Omron CX-Programmer project NuevoProyecto (CX-Programmer 9.31)

# PLC NuevoPLC1: CJ1M CPU11

## Program NuevoPrograma1 (cyclic task 0)
; La v1.1 funciona correctament la inicialitzacio, manual(La linea 1 del E_F4 te un SMM ja que sino al sortir es mantidria EM_0 en on)
Local symbols
C1_BE 0.07 BOOL  ; Bolet de emergencia
C1_COM1_FI_CUA W511.02 BOOL  ; CUADRAT  COMPLETS COMANDA 1
C1_COM1_FI_PEN W511.03 BOOL  ; PENTAGO COMPLETS COMANDA 1
C1_COM1_FI_ROD W511.01 BOOL  ; RODONA COMPLETS COMANDA 1
C1_COM1_FI_TRI W511.00 BOOL  ; TRIANGLES COMPLETS COMANDA 1
C1_COM2_FI_CUA W511.06 BOOL  ; CUADRAT COMPLETS COMANDA 2
C1_COM2_FI_PEN W511.07 BOOL  ; PENTAGON COMPLETS COMANDA 2
C1_COM2_FI_ROD W511.05 BOOL  ; RODONA COMPLETS COMANDA 2
C1_COM2_FI_TRI W511.04 BOOL  ; TRIANGLES COMPLETS COMANDA 2
C1_DET1 0.09 BOOL  ; Detector 1 cinta 1
C1_DET2 0.08 BOOL  ; Detector 2 cinta 1
C1_DET3 0.10 BOOL  ; Detector 3 cinta 1
C1_DET4 0.11 BOOL  ; Detector 4 cinta 1
C1_EA_0 W300.00 BOOL  ; Etapa automatic 0
C1_EA_1 W300.01 BOOL  ; Etapa automatica 1 MFW
C1_EA_10 W300.10 BOOL  ; COMANDA 2 TRIANGLE ++
C1_EA_11 W300.11 BOOL  ; TRIANGLE A REBUIG
C1_EA_18 W300.12 BOOL  ; Etapa automatica 18 cuadrat
C1_EA_19 W300.13 BOOL  ; COMANDA 1 CUADRAT ++
C1_EA_2 W300.02 BOOL  ; Etapa automatica 2 T1
C1_EA_20 W300.14 BOOL  ; COMANDA 2 CUADRAT ++
C1_EA_21 W300.15 BOOL  ; CUADRAT REBUIG
C1_EA_28 W301.00 BOOL  ; ETAPA AUTOMATIC 28 PENTAGON
C1_EA_29 W301.01 BOOL  ; COMANDA 1 PENTAGON ++
C1_EA_3 W300.03 BOOL  ; Etapa automatica 3 MOFF
C1_EA_30 W301.02 BOOL  ; COMANDA 2 PENTAGON++
C1_EA_31 W301.03 BOOL  ; PENTAGON REBUIG
C1_EA_38 W301.04 BOOL  ; ESTAPA AUTOMATIC 38 RODONA
C1_EA_39 W301.05 BOOL  ; COMANDA 1 RODONA ++
C1_EA_4 W300.04 BOOL  ; Etapa automatica 4 NO EVA 1
C1_EA_40 W301.06 BOOL  ; COMANDA 2 RODONA ++
C1_EA_41 W301.07 BOOL  ; RODONA REBUIG
C1_EA_42 W301.08 BOOL  ; FI CICLE
C1_EA_5 W300.05 BOOL  ; Etapa automatica 5 OK EVA
C1_EA_6 W300.06 BOOL  ; Etapa automatica 6 T2
C1_EA_7 W300.07 BOOL  ; Etapa automatica DET4
C1_EA_8 W300.08 BOOL  ; Etapa automatica 8 Triangle
C1_EA_9 W300.09 BOOL  ; COMANDA 1 TRIANGLE++
C1_EM_0 W200.00 BOOL  ; Etapa 0 Manual
C1_EM_1 W200.01 BOOL  ; Etapa Manual1-Motor Forware
C1_EM_2 W200.02 BOOL  ; Etapa Manual2-Motor Reware
C1_EM_3 W200.03 BOOL  ; Etapa manual 3 - Aturada motor
C1_E_A1 W400.00 BOOL
C1_E_A2 W400.03 BOOL  ; Parada solicitud final de cicle
C1_E_D1 W400.05 BOOL  ; Parada de emergencia
C1_E_D3 W400.06 BOOL  ; Parada postemergencia
C1_E_F1 W400.01 BOOL  ; Produccio normal
C1_E_F4 W400.02 BOOL  ; Marcha de verificacio sense ordre
C1_E_F41 W400.04 BOOL  ; Etapa de pas Sortida Manual
C1_E_F6 W400.07 BOOL  ; Teach Marxa de Test
C1_E_F61 W400.08 BOOL  ; Teach 2
C1_HMI_A1 W103.00 BOOL  ; HABILITACIO A SCADA DE E_A1
C1_HMI_A6 W103.03 BOOL  ; HABILITACIO A SCADA DE A6
C1_HMI_COM1_PEN W14 CHANNEL  ; ENVIA EL ESTAT DE PENTAGON DE COMANDA 1
C1_HMI_COM1_QUA W12 CHANNEL  ; ENVIA EL ESTAT DE CUADRATS DE COMANDA 1
C1_HMI_COM1_ROD W13 CHANNEL  ; ENVIA EL ESTAT DE RODONES DE COMANDA 1
C1_HMI_COM1_TRI W11 CHANNEL  ; ENVIA EL ESTAT DE TRIANGLES DE COMANDA 1
C1_HMI_COM2_PEN W18 CHANNEL  ; ENVIA EL ESTAT DE PENTAGO  DE COMANDA 2
C1_HMI_COM2_QUA W16 CHANNEL  ; ENVIA EL ESTAT DE CUADRAT DE COMANDA 2
C1_HMI_COM2_ROD W17 CHANNEL  ; ENVIA EL ESTAT DE RODONA DE COMANDA 2
C1_HMI_COM2_TRI W15 CHANNEL  ; ENVIA EL ESTAT DE TRIANGLES DE COMANDA 2
C1_HMI_D2 W103.04 BOOL  ; HABILITACIO A SCADA DE D1
C1_HMI_EMER_FIS W101.03 BOOL  ; AVIS DE CINTA DE EMERGENCIA FISICA
C1_HMI_EMER_LOG W101.02 BOOL  ; AVIS CINTA DE EMERGENCIA LOGICA
C1_HMI_F1 W103.01 BOOL  ; HABILITACIO A SCADA DE F1
C1_HMI_F4 W103.02 BOOL  ; HABILITACIO A SCADA DE F4
C1_HMI_MOT_OK W101.00 BOOL  ; AVIS A LA HMI QUE LA CINTA FUNCIONA
C1_HMI_PR W101.04 BOOL  ; AVIS DEL POLSADOR DE REARME A HMI
C1_H_AMB 1.09 BOOL
C1_H_AUTO 1.03 BOOL
C1_H_MANUAL 1.04 BOOL
C1_H_ROJ 1.10 BOOL
C1_H_TEACH 1.05 BOOL
C1_H_VER 1.08 BOOL
C1_JFW 0.06 BOOL  ; Joystick Forware
C1_JRW 0.05 BOOL  ; Joystick Reward
C1_KA10 1.07 BOOL
C1_KA9 1.06 BOOL
C1_MF W201.00 BOOL  ; Marca First scan
C1_MFW 1.01 BOOL  ; Motor Forward
C1_MM W100.15 BOOL  ; Marca marxa
C1_MPP W201.04 BOOL  ; MARCA DE PARO
C1_MRW 1.00 BOOL  ; Motor Reward
C1_NOK_EVA W501.00 BOOL  ; Foto erronea
C1_OK_EVA 500.02 BOOL  ; Foto correcta
C1_PM 0.02 BOOL  ; Polsador marxa
C1_PP 0.03 BOOL  ; Polsador paro
C1_PR 0.04 BOOL  ; Polsador rearme
C1_REP W501.01 BOOL  ; Repetir foto
C1_SM1 0.00 BOOL  ; Selector de mode Pos.1
C1_SM2 0.01 BOOL  ; Selector de mode Pos.2
C1_SMA W201.01 BOOL  ; Marca selector automatic
C1_SMM 201.02 BOOL  ; Marca selector manual
C1_SMT 201.03 BOOL  ; Marca selector Teach
C1_TEACH_OK H0.00 BOOL  ; Captura correcte peça
C2_FI_CICLE 3101.00 BOOL
C2_MAGATZEM_1_3 3100.00 BOOL
C2_MAGATZEM_2_4 3100.01 BOOL
COMP_PEN1 W100.04 BOOL  ; COMPARA PENTAGONS COM1
COMP_PEN2 W100.05 BOOL  ; COMPARA PENTAGONS COM2
COMP_QUA1 W100.02 BOOL  ; COMPARA QUADRATS COM1
COMP_QUA2 W100.03 BOOL  ; COMPARA QUADRATS COM2
COMP_ROD1 W100.06 BOOL  ; COMPARA RODONES COM1
COMP_ROD2 W100.07 BOOL  ; COMPARA RODONES COM2
COMP_TRI1 W100.00 BOOL  ; COMPARA TRIANGLES COM1
COMP_TRI2 W100.01 BOOL  ; COMPARA TRIANGLES COM2
CUA_COM1 W305.02 BOOL
CUA_COM2 W305.03 BOOL
EVA_CUADRAT W510.01 BOOL  ; Foto per EVA=CUADRAT
EVA_ENABLE 510.04 BOOL  ; ACTIVAR EVA
EVA_PENTAGON W510.03 BOOL  ; Foto per EVA=PENTAGON
EVA_RODONA W510.02 BOOL  ; Foto per EVA=RODONA
EVA_TRIANGLE W510.00 BOOL  ; Foto per EVA=TRIANGLE
HMI_BE W101.05 BOOL  ; BOLET DE EMERGENCIA HMI
HMI_C1_COM1_OK W101.13 BOOL  ; VALIDACIO COM 1
HMI_C1_COM2_OK W101.14 BOOL  ; VALIDACIO COM2
HMI_C1_JF W101.08 BOOL  ; HMI C1 JOYSTICKDRETA
HMI_C1_JR W101.09 BOOL  ; HMI C1 JOYSTIC REWARD
HMI_C1_PSW W101.15 BOOL  ; PASSWORD OK
HMI_C1_Q_NO W102.01 BOOL  ; RESPOSTA NEGATIVA A ACABAR CICLE
HMI_C1_Q_SI W102.00 BOOL  ; RESPOSTA AFIRMATIVA A ACABAR CICLE
HMI_C1_TEMP_DET3 W10 UINT_BCD  ; TEMPORITZADOR DET3-DET4
HMI_C1_TEMP_EVA W9 UINT_BCD  ; TEMPORTIZADOR EVA
HMI_COM1_CUA W1 CHANNEL  ; DEMANDA DE CUADRATS PER COMANDA 1
HMI_COM1_PEN W2 CHANNEL  ; DEMANDA DE PENTAGON PER COMANDA 1
HMI_COM1_ROD W3 CHANNEL  ; DEMANDA DE RODONA PER COMANDA 1
HMI_COM1_TRI W4 CHANNEL  ; DEMANDA DE TRIANGLE PER COMANDA 1
HMI_COM2_CUA W5 CHANNEL  ; DEMANDA DE CUADRATS PER COMANDA 2
HMI_COM2_PEN W6 CHANNEL  ; DEMANDA DE PENTAGON PER COMANDA 2
HMI_COM2_ROD W7 CHANNEL  ; DEMANDA DE RODONA PER COMANDA 2
HMI_COM2_TRI W8 CHANNEL  ; DEMANDA DE TRIANGLE PER COMANDA 2
HMI_EMER_OK W101.12 BOOL  ; Validacio de emerencies
HMI_PM W101.07 BOOL  ; Polsador de marxa des de HMI
HMI_PP W101.06 BOOL  ; Polsador de paro des de HMI
MAN_FWD W201.02 BOOL  ; MOTOR FORDWARD MANUAL
MAN_RWD W201.03 BOOL  ; MOTOR REWARD MANUAL
PEN_COM1 W305.04 BOOL
PEN_COM2 W305.05 BOOL
ROD_COM1 W305.06 BOOL
ROD_COM2 W305.07 BOOL
TRI_COM1 W305.00 BOOL
TRI_COM2 W305.01 BOOL

### Section INICIALITZACIÓ_I_ETAPA_ACTIVA_GEMMA

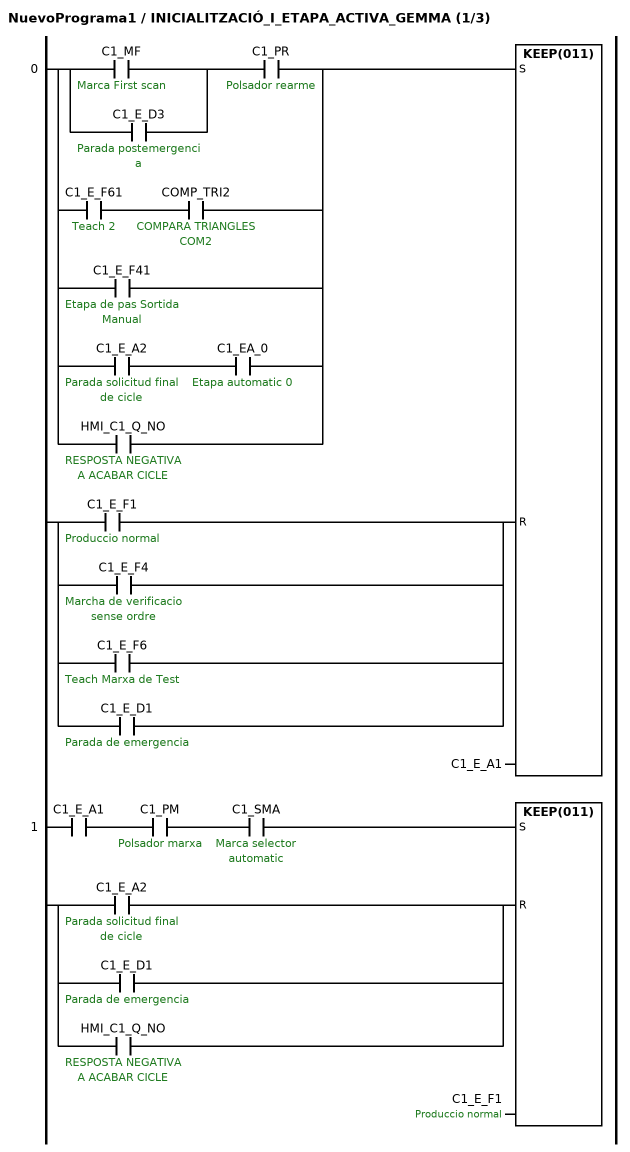
; rung 0
LD C1_MF  ; Marca First scan
OR C1_E_D3  ; Parada postemergencia
AND C1_PR  ; Polsador rearme
LD C1_E_F61  ; Teach 2
AND COMP_TRI2  ; COMPARA TRIANGLES COM2
ORLD
OR C1_E_F41  ; Etapa de pas Sortida Manual
LD C1_E_A2  ; Parada solicitud final de cicle
AND C1_EA_0  ; Etapa automatic 0
ORLD
OR HMI_C1_Q_NO  ; RESPOSTA NEGATIVA A ACABAR CICLE
LD C1_E_F1  ; Produccio normal
OR C1_E_F4  ; Marcha de verificacio sense ordre
OR C1_E_F6  ; Teach Marxa de Test
OR C1_E_D1  ; Parada de emergencia
KEEP(011) C1_E_A1
; rung 1
LD C1_E_A1
AND C1_PM  ; Polsador marxa
AND C1_SMA  ; Marca selector automatic
LD C1_E_A2  ; Parada solicitud final de cicle
OR C1_E_D1  ; Parada de emergencia
OR HMI_C1_Q_NO  ; RESPOSTA NEGATIVA A ACABAR CICLE
KEEP(011) C1_E_F1  ; Produccio normal

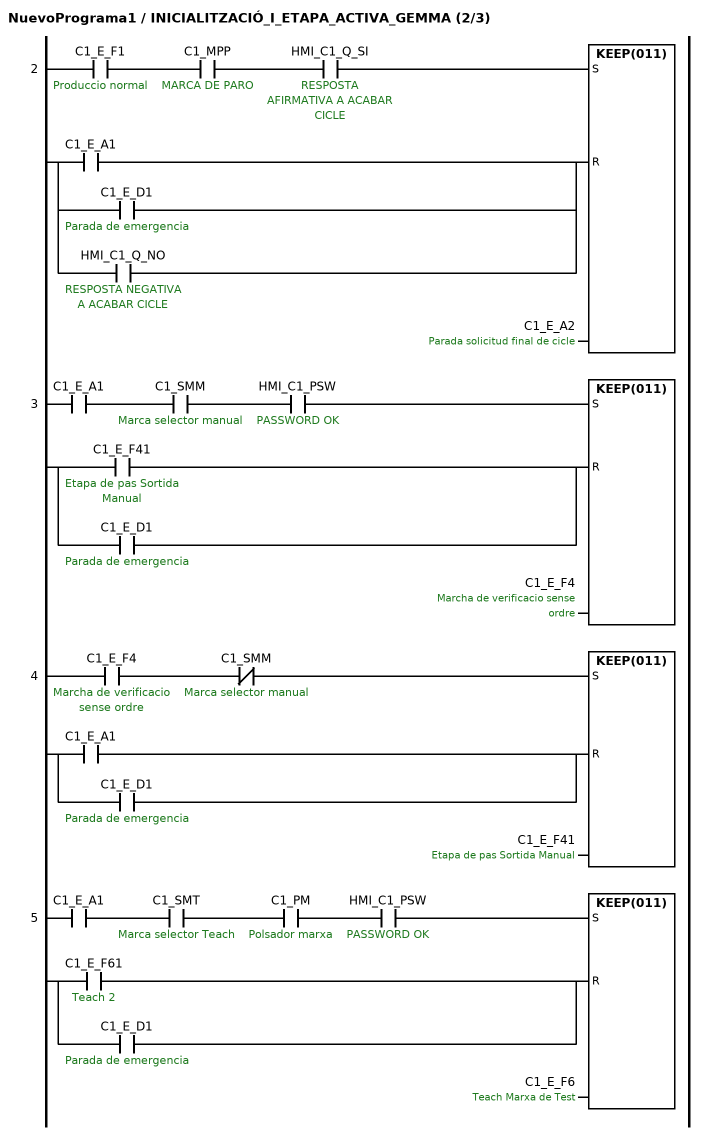
; rung 2
LD C1_E_F1  ; Produccio normal
AND C1_MPP  ; MARCA DE PARO
AND HMI_C1_Q_SI  ; RESPOSTA AFIRMATIVA A ACABAR CICLE
LD C1_E_A1
OR C1_E_D1  ; Parada de emergencia
OR HMI_C1_Q_NO  ; RESPOSTA NEGATIVA A ACABAR CICLE
KEEP(011) C1_E_A2  ; Parada solicitud final de cicle
; rung 3
LD C1_E_A1
AND C1_SMM  ; Marca selector manual
AND HMI_C1_PSW  ; PASSWORD OK
LD C1_E_F41  ; Etapa de pas Sortida Manual
OR C1_E_D1  ; Parada de emergencia
KEEP(011) C1_E_F4  ; Marcha de verificacio sense ordre
; rung 4
LD C1_E_F4  ; Marcha de verificacio sense ordre
ANDNOT C1_SMM  ; Marca selector manual
LD C1_E_A1
OR C1_E_D1  ; Parada de emergencia
KEEP(011) C1_E_F41  ; Etapa de pas Sortida Manual
; rung 5
LD C1_E_A1
AND C1_SMT  ; Marca selector Teach
AND C1_PM  ; Polsador marxa
AND HMI_C1_PSW  ; PASSWORD OK
LD C1_E_F61  ; Teach 2
OR C1_E_D1  ; Parada de emergencia
KEEP(011) C1_E_F6  ; Teach Marxa de Test

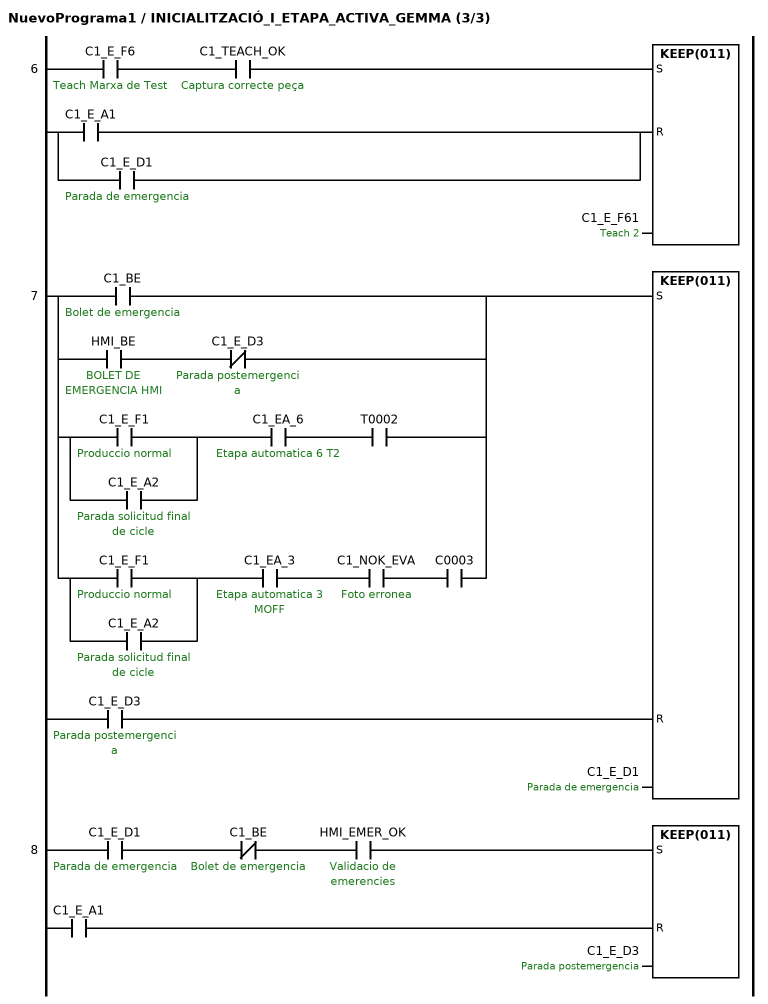
; rung 6
LD C1_E_F6  ; Teach Marxa de Test
AND C1_TEACH_OK  ; Captura correcte peça
LD C1_E_A1
OR C1_E_D1  ; Parada de emergencia
KEEP(011) C1_E_F61  ; Teach 2
; rung 7
LD C1_BE  ; Bolet de emergencia
LD HMI_BE  ; BOLET DE EMERGENCIA HMI
ANDNOT C1_E_D3  ; Parada postemergencia
ORLD
LD C1_E_F1  ; Produccio normal
OR C1_E_A2  ; Parada solicitud final de cicle
AND C1_EA_6  ; Etapa automatica 6 T2
AND T0002
ORLD
LD C1_E_F1  ; Produccio normal
OR C1_E_A2  ; Parada solicitud final de cicle
AND C1_EA_3  ; Etapa automatica 3 MOFF
AND C1_NOK_EVA  ; Foto erronea
AND C0003
ORLD
LD C1_E_D3  ; Parada postemergencia
KEEP(011) C1_E_D1  ; Parada de emergencia
; rung 8
LD C1_E_D1  ; Parada de emergencia
ANDNOT C1_BE  ; Bolet de emergencia
AND HMI_EMER_OK  ; Validacio de emerencies
LD C1_E_A1
KEEP(011) C1_E_D3  ; Parada postemergencia

### Section ACCIONS_GEMMA

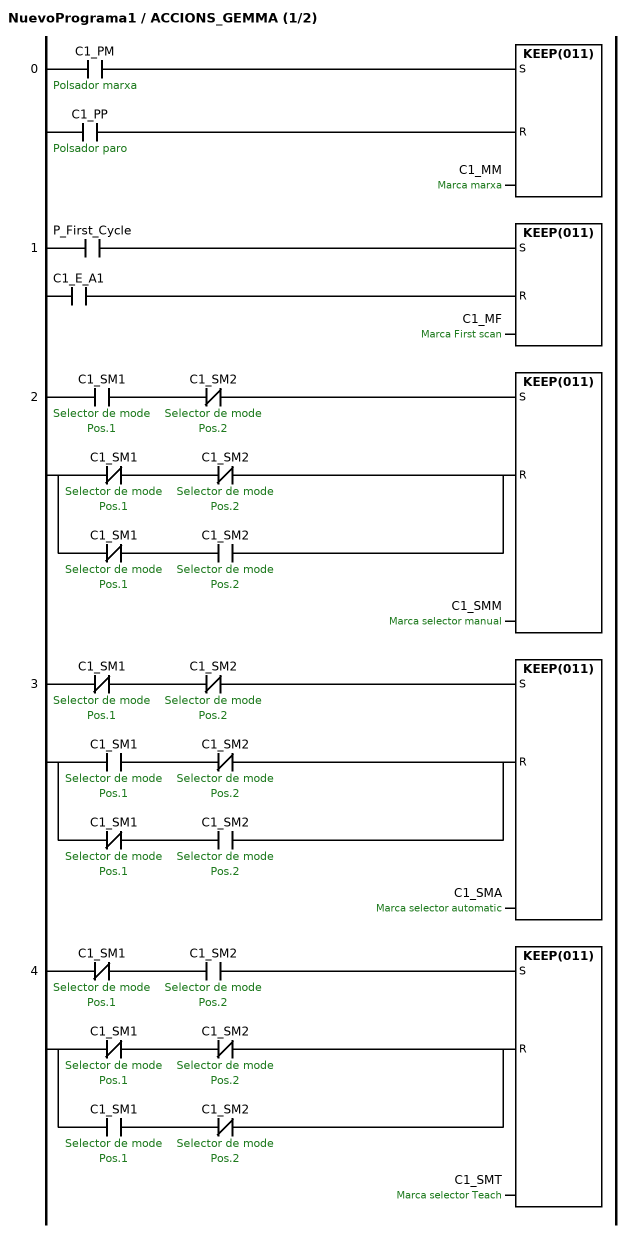
; rung 0
LD C1_PM  ; Polsador marxa
LD C1_PP  ; Polsador paro
KEEP(011) C1_MM  ; Marca marxa
; rung 1
LD P_First_Cycle
LD C1_E_A1
KEEP(011) C1_MF  ; Marca First scan
; rung 2
LD C1_SM1  ; Selector de mode Pos.1
ANDNOT C1_SM2  ; Selector de mode Pos.2
LDNOT C1_SM1  ; Selector de mode Pos.1
ANDNOT C1_SM2  ; Selector de mode Pos.2
LDNOT C1_SM1  ; Selector de mode Pos.1
AND C1_SM2  ; Selector de mode Pos.2
ORLD
KEEP(011) C1_SMM  ; Marca selector manual
; rung 3
LDNOT C1_SM1  ; Selector de mode Pos.1
ANDNOT C1_SM2  ; Selector de mode Pos.2
LD C1_SM1  ; Selector de mode Pos.1
ANDNOT C1_SM2  ; Selector de mode Pos.2
LDNOT C1_SM1  ; Selector de mode Pos.1
AND C1_SM2  ; Selector de mode Pos.2
ORLD
KEEP(011) C1_SMA  ; Marca selector automatic
; rung 4
LDNOT C1_SM1  ; Selector de mode Pos.1
AND C1_SM2  ; Selector de mode Pos.2
LDNOT C1_SM1  ; Selector de mode Pos.1
ANDNOT C1_SM2  ; Selector de mode Pos.2
LD C1_SM1  ; Selector de mode Pos.1
ANDNOT C1_SM2  ; Selector de mode Pos.2
ORLD
KEEP(011) C1_SMT  ; Marca selector Teach

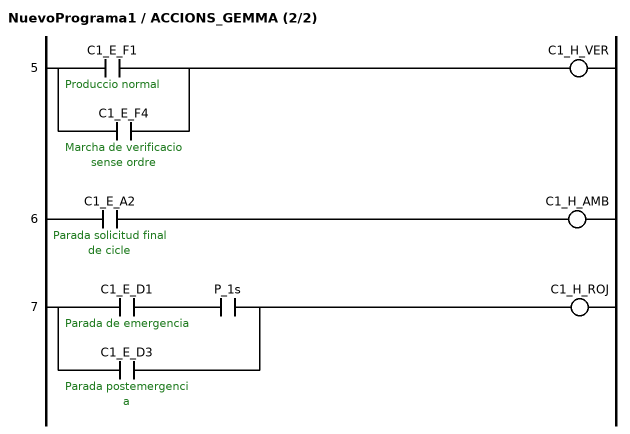
; rung 5
LD C1_E_F1  ; Produccio normal
OR C1_E_F4  ; Marcha de verificacio sense ordre
OUT C1_H_VER
; rung 6
LD C1_E_A2  ; Parada solicitud final de cicle
OUT C1_H_AMB
; rung 7
LD C1_E_D1  ; Parada de emergencia
AND P_1s
OR C1_E_D3  ; Parada postemergencia
OUT C1_H_ROJ

### Section E_F1

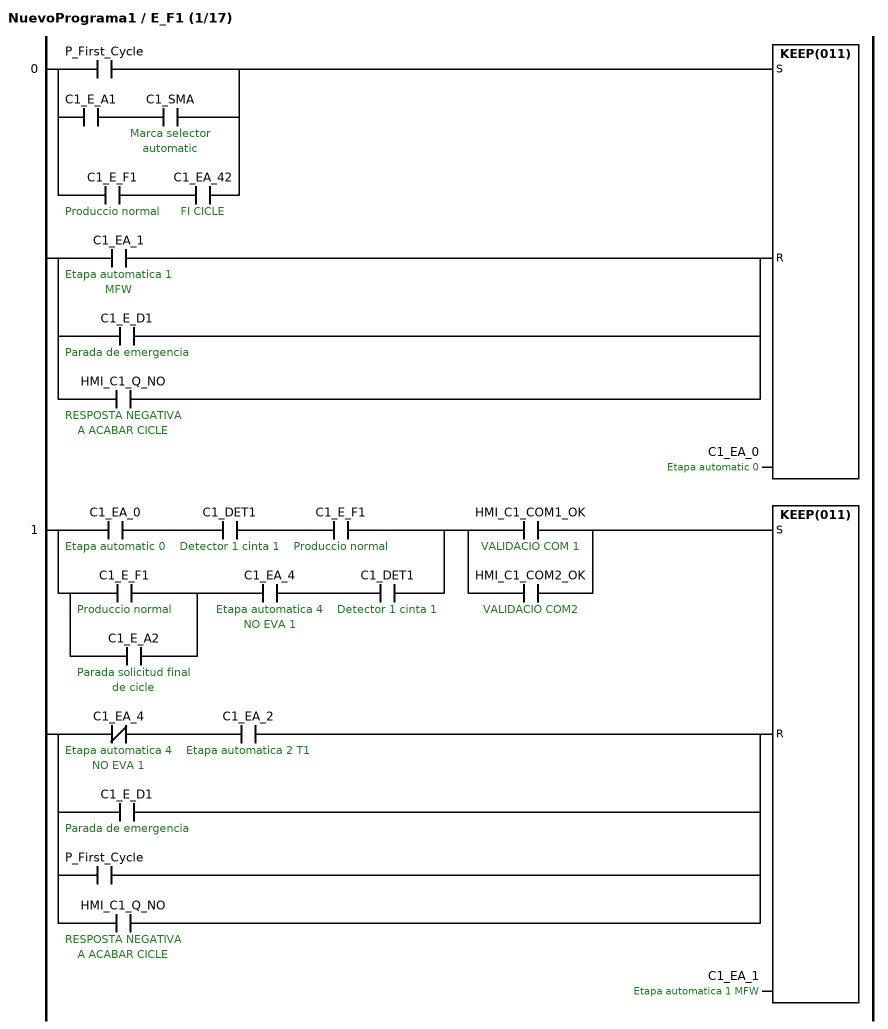
; rung 0
LD P_First_Cycle
LD C1_E_A1
AND C1_SMA  ; Marca selector automatic
ORLD
LD C1_E_F1  ; Produccio normal
AND C1_EA_42  ; FI CICLE
ORLD
LD C1_EA_1  ; Etapa automatica 1 MFW
OR C1_E_D1  ; Parada de emergencia
OR HMI_C1_Q_NO  ; RESPOSTA NEGATIVA A ACABAR CICLE
KEEP(011) C1_EA_0  ; Etapa automatic 0
; rung 1
LD C1_EA_0  ; Etapa automatic 0
AND C1_DET1  ; Detector 1 cinta 1
AND C1_E_F1  ; Produccio normal
LD C1_E_F1  ; Produccio normal
OR C1_E_A2  ; Parada solicitud final de cicle
AND C1_EA_4  ; Etapa automatica 4 NO EVA 1
AND C1_DET1  ; Detector 1 cinta 1
ORLD
LD HMI_C1_COM1_OK  ; VALIDACIO COM 1
OR HMI_C1_COM2_OK  ; VALIDACIO COM2
ANDLD
LDNOT C1_EA_4  ; Etapa automatica 4 NO EVA 1
AND C1_EA_2  ; Etapa automatica 2 T1
OR C1_E_D1  ; Parada de emergencia
OR P_First_Cycle
OR HMI_C1_Q_NO  ; RESPOSTA NEGATIVA A ACABAR CICLE
KEEP(011) C1_EA_1  ; Etapa automatica 1 MFW

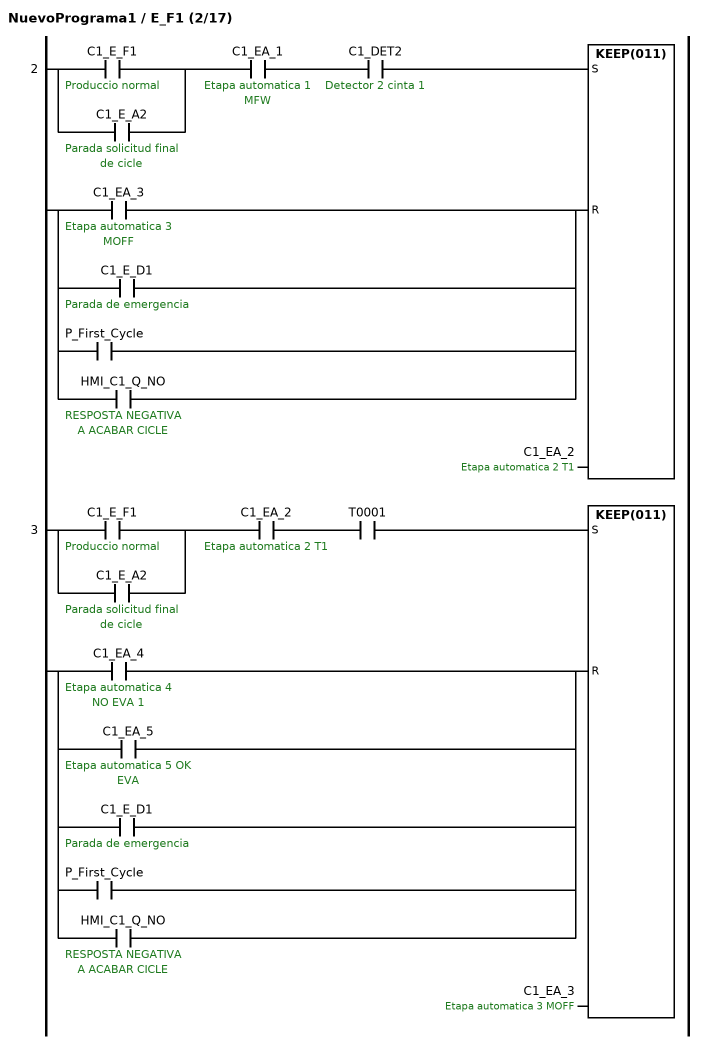
; rung 2
LD C1_E_F1  ; Produccio normal
OR C1_E_A2  ; Parada solicitud final de cicle
AND C1_EA_1  ; Etapa automatica 1 MFW
AND C1_DET2  ; Detector 2 cinta 1
LD C1_EA_3  ; Etapa automatica 3 MOFF
OR C1_E_D1  ; Parada de emergencia
OR P_First_Cycle
OR HMI_C1_Q_NO  ; RESPOSTA NEGATIVA A ACABAR CICLE
KEEP(011) C1_EA_2  ; Etapa automatica 2 T1
; rung 3
LD C1_E_F1  ; Produccio normal
OR C1_E_A2  ; Parada solicitud final de cicle
AND C1_EA_2  ; Etapa automatica 2 T1
AND T0001
LD C1_EA_4  ; Etapa automatica 4 NO EVA 1
OR C1_EA_5  ; Etapa automatica 5 OK EVA
OR C1_E_D1  ; Parada de emergencia
OR P_First_Cycle
OR HMI_C1_Q_NO  ; RESPOSTA NEGATIVA A ACABAR CICLE
KEEP(011) C1_EA_3  ; Etapa automatica 3 MOFF

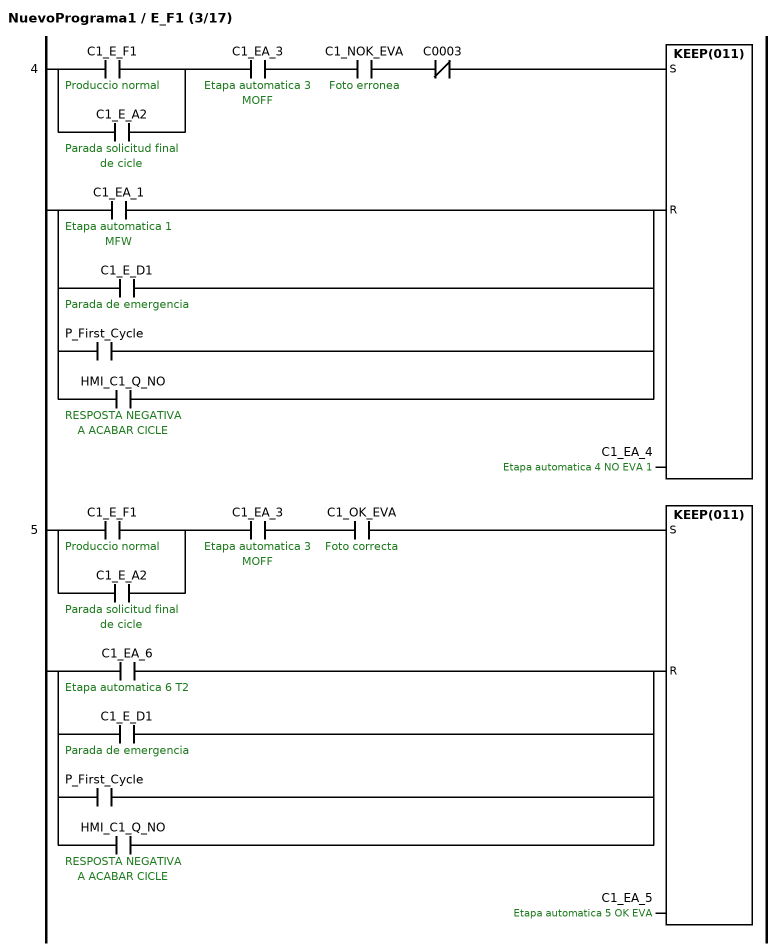
; rung 4
LD C1_E_F1  ; Produccio normal
OR C1_E_A2  ; Parada solicitud final de cicle
AND C1_EA_3  ; Etapa automatica 3 MOFF
AND C1_NOK_EVA  ; Foto erronea
ANDNOT C0003
LD C1_EA_1  ; Etapa automatica 1 MFW
OR C1_E_D1  ; Parada de emergencia
OR P_First_Cycle
OR HMI_C1_Q_NO  ; RESPOSTA NEGATIVA A ACABAR CICLE
KEEP(011) C1_EA_4  ; Etapa automatica 4 NO EVA 1
; rung 5
LD C1_E_F1  ; Produccio normal
OR C1_E_A2  ; Parada solicitud final de cicle
AND C1_EA_3  ; Etapa automatica 3 MOFF
AND C1_OK_EVA  ; Foto correcta
LD C1_EA_6  ; Etapa automatica 6 T2
OR C1_E_D1  ; Parada de emergencia
OR P_First_Cycle
OR HMI_C1_Q_NO  ; RESPOSTA NEGATIVA A ACABAR CICLE
KEEP(011) C1_EA_5  ; Etapa automatica 5 OK EVA

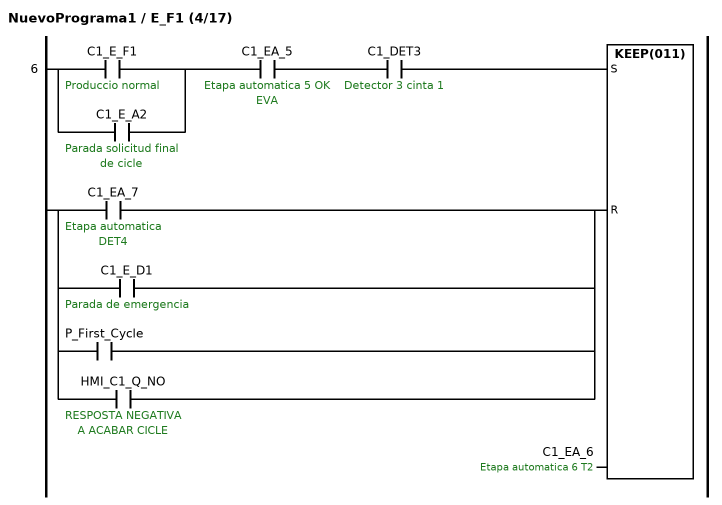
; rung 6
LD C1_E_F1  ; Produccio normal
OR C1_E_A2  ; Parada solicitud final de cicle
AND C1_EA_5  ; Etapa automatica 5 OK EVA
AND C1_DET3  ; Detector 3 cinta 1
LD C1_EA_7  ; Etapa automatica DET4
OR C1_E_D1  ; Parada de emergencia
OR P_First_Cycle
OR HMI_C1_Q_NO  ; RESPOSTA NEGATIVA A ACABAR CICLE
KEEP(011) C1_EA_6  ; Etapa automatica 6 T2

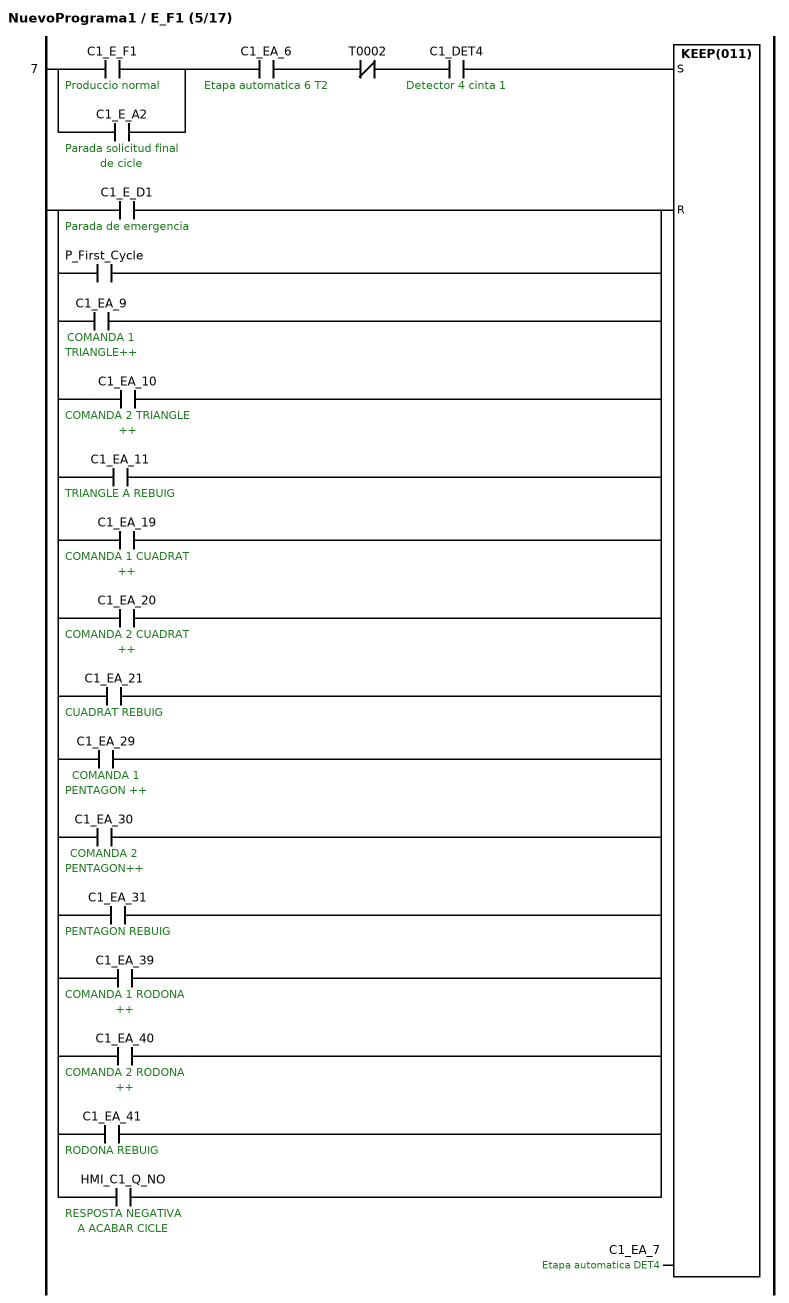
; rung 7
LD C1_E_F1  ; Produccio normal
OR C1_E_A2  ; Parada solicitud final de cicle
AND C1_EA_6  ; Etapa automatica 6 T2
ANDNOT T0002
AND C1_DET4  ; Detector 4 cinta 1
LD C1_E_D1  ; Parada de emergencia
OR P_First_Cycle
OR C1_EA_9  ; COMANDA 1 TRIANGLE++
OR C1_EA_10  ; COMANDA 2 TRIANGLE ++
OR C1_EA_11  ; TRIANGLE A REBUIG
OR C1_EA_19  ; COMANDA 1 CUADRAT ++
OR C1_EA_20  ; COMANDA 2 CUADRAT ++
OR C1_EA_21  ; CUADRAT REBUIG
OR C1_EA_29  ; COMANDA 1 PENTAGON ++
OR C1_EA_30  ; COMANDA 2 PENTAGON++
OR C1_EA_31  ; PENTAGON REBUIG
OR C1_EA_39  ; COMANDA 1 RODONA ++
OR C1_EA_40  ; COMANDA 2 RODONA ++
OR C1_EA_41  ; RODONA REBUIG
OR HMI_C1_Q_NO  ; RESPOSTA NEGATIVA A ACABAR CICLE
KEEP(011) C1_EA_7  ; Etapa automatica DET4

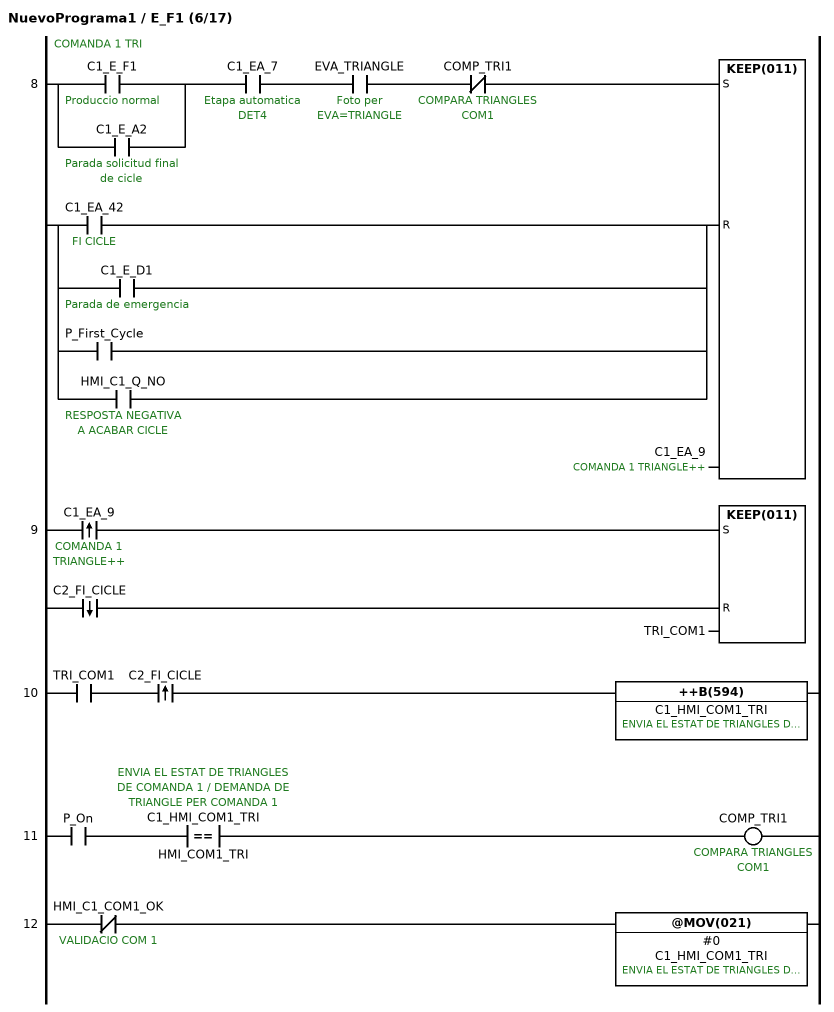
; rung 8: COMANDA 1 TRI
LD C1_E_F1  ; Produccio normal
OR C1_E_A2  ; Parada solicitud final de cicle
AND C1_EA_7  ; Etapa automatica DET4
AND EVA_TRIANGLE  ; Foto per EVA=TRIANGLE
ANDNOT COMP_TRI1  ; COMPARA TRIANGLES COM1
LD C1_EA_42  ; FI CICLE
OR C1_E_D1  ; Parada de emergencia
OR P_First_Cycle
OR HMI_C1_Q_NO  ; RESPOSTA NEGATIVA A ACABAR CICLE
KEEP(011) C1_EA_9  ; COMANDA 1 TRIANGLE++
; rung 9
@LD C1_EA_9  ; COMANDA 1 TRIANGLE++
%LD C2_FI_CICLE
KEEP(011) TRI_COM1
; rung 10
LD TRI_COM1
@AND C2_FI_CICLE
++B(594) C1_HMI_COM1_TRI  ; ENVIA EL ESTAT DE TRIANGLES DE COMANDA 1
; rung 11
LD P_On
AND=(300) C1_HMI_COM1_TRI HMI_COM1_TRI  ; ENVIA EL ESTAT DE TRIANGLES DE COMANDA 1, DEMANDA DE TRIANGLE PER COMANDA 1
OUT COMP_TRI1  ; COMPARA TRIANGLES COM1
; rung 12
LDNOT HMI_C1_COM1_OK  ; VALIDACIO COM 1
@MOV(021) #0 C1_HMI_COM1_TRI  ; ENVIA EL ESTAT DE TRIANGLES DE COMANDA 1

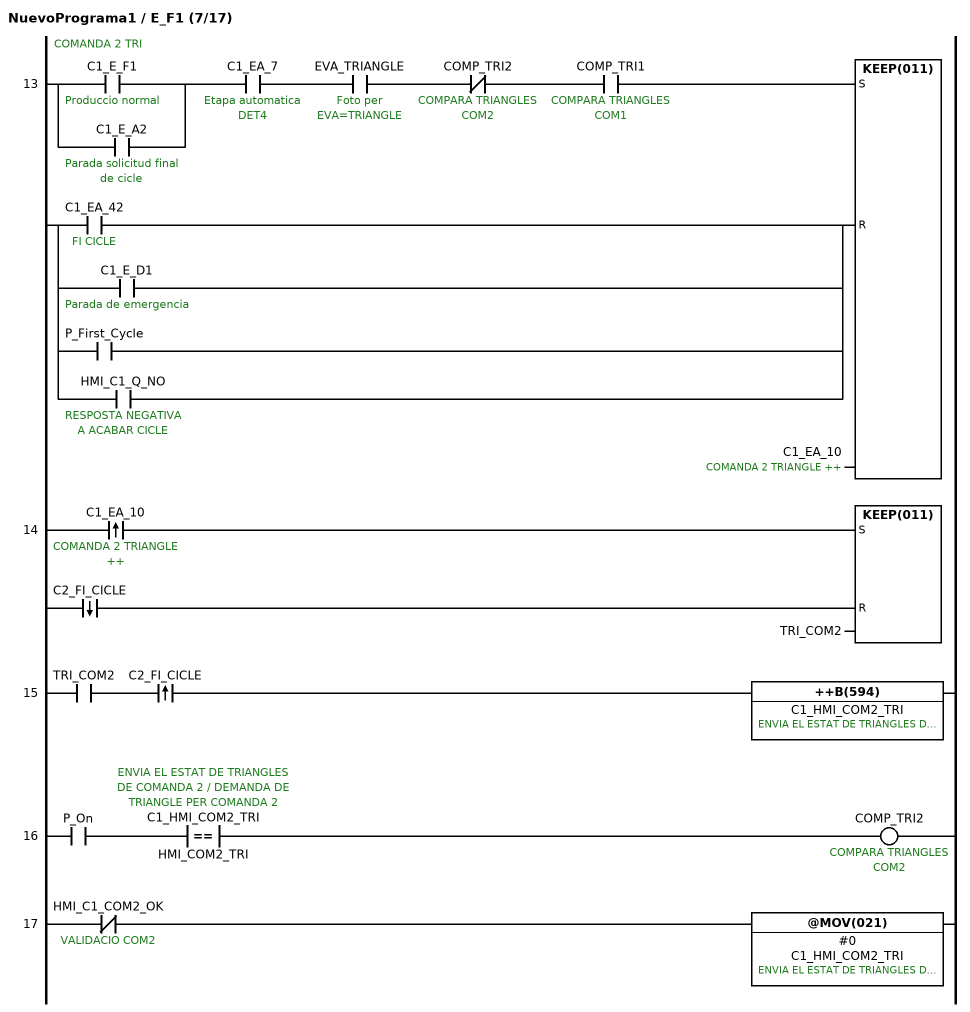
; rung 13: COMANDA 2 TRI
LD C1_E_F1  ; Produccio normal
OR C1_E_A2  ; Parada solicitud final de cicle
AND C1_EA_7  ; Etapa automatica DET4
AND EVA_TRIANGLE  ; Foto per EVA=TRIANGLE
ANDNOT COMP_TRI2  ; COMPARA TRIANGLES COM2
AND COMP_TRI1  ; COMPARA TRIANGLES COM1
LD C1_EA_42  ; FI CICLE
OR C1_E_D1  ; Parada de emergencia
OR P_First_Cycle
OR HMI_C1_Q_NO  ; RESPOSTA NEGATIVA A ACABAR CICLE
KEEP(011) C1_EA_10  ; COMANDA 2 TRIANGLE ++
; rung 14
@LD C1_EA_10  ; COMANDA 2 TRIANGLE ++
%LD C2_FI_CICLE
KEEP(011) TRI_COM2
; rung 15
LD TRI_COM2
@AND C2_FI_CICLE
++B(594) C1_HMI_COM2_TRI  ; ENVIA EL ESTAT DE TRIANGLES DE COMANDA 2
; rung 16
LD P_On
AND=(300) C1_HMI_COM2_TRI HMI_COM2_TRI  ; ENVIA EL ESTAT DE TRIANGLES DE COMANDA 2, DEMANDA DE TRIANGLE PER COMANDA 2
OUT COMP_TRI2  ; COMPARA TRIANGLES COM2
; rung 17
LDNOT HMI_C1_COM2_OK  ; VALIDACIO COM2
@MOV(021) #0 C1_HMI_COM2_TRI  ; ENVIA EL ESTAT DE TRIANGLES DE COMANDA 2

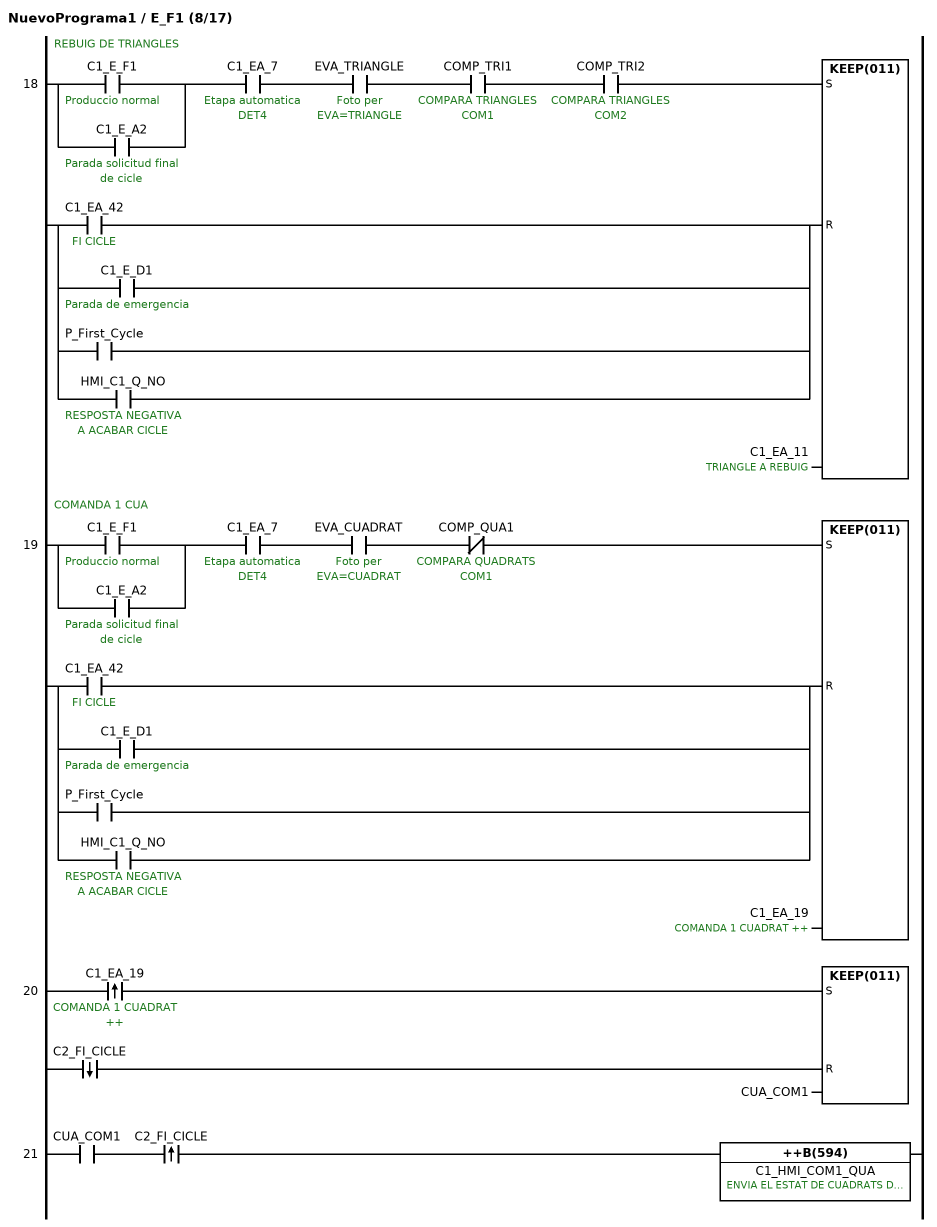
; rung 18: REBUIG DE TRIANGLES
LD C1_E_F1  ; Produccio normal
OR C1_E_A2  ; Parada solicitud final de cicle
AND C1_EA_7  ; Etapa automatica DET4
AND EVA_TRIANGLE  ; Foto per EVA=TRIANGLE
AND COMP_TRI1  ; COMPARA TRIANGLES COM1
AND COMP_TRI2  ; COMPARA TRIANGLES COM2
LD C1_EA_42  ; FI CICLE
OR C1_E_D1  ; Parada de emergencia
OR P_First_Cycle
OR HMI_C1_Q_NO  ; RESPOSTA NEGATIVA A ACABAR CICLE
KEEP(011) C1_EA_11  ; TRIANGLE A REBUIG
; rung 19: COMANDA 1 CUA
LD C1_E_F1  ; Produccio normal
OR C1_E_A2  ; Parada solicitud final de cicle
AND C1_EA_7  ; Etapa automatica DET4
AND EVA_CUADRAT  ; Foto per EVA=CUADRAT
ANDNOT COMP_QUA1  ; COMPARA QUADRATS COM1
LD C1_EA_42  ; FI CICLE
OR C1_E_D1  ; Parada de emergencia
OR P_First_Cycle
OR HMI_C1_Q_NO  ; RESPOSTA NEGATIVA A ACABAR CICLE
KEEP(011) C1_EA_19  ; COMANDA 1 CUADRAT ++
; rung 20
@LD C1_EA_19  ; COMANDA 1 CUADRAT ++
%LD C2_FI_CICLE
KEEP(011) CUA_COM1
; rung 21
LD CUA_COM1
@AND C2_FI_CICLE
++B(594) C1_HMI_COM1_QUA  ; ENVIA EL ESTAT DE CUADRATS DE COMANDA 1

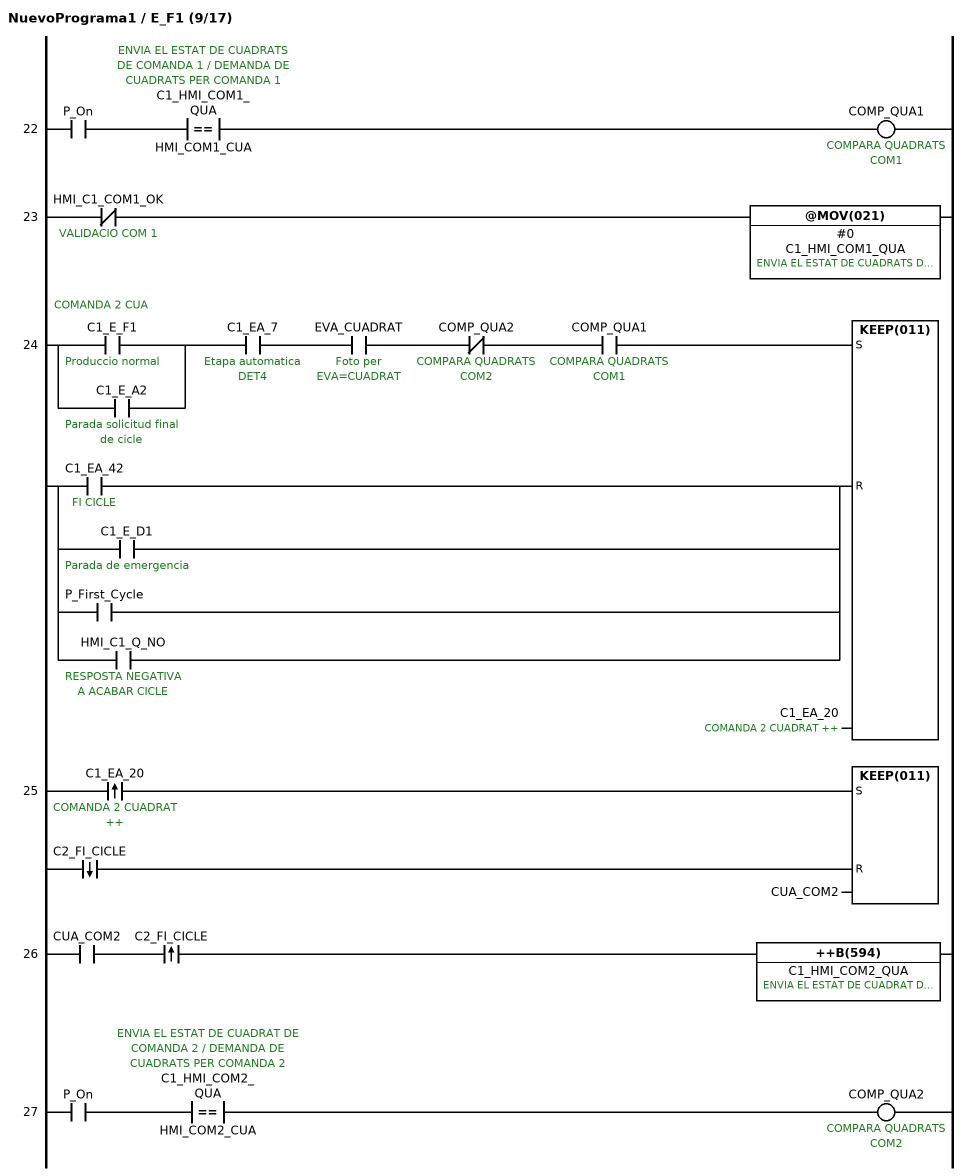
; rung 22
LD P_On
AND=(300) C1_HMI_COM1_QUA HMI_COM1_CUA  ; ENVIA EL ESTAT DE CUADRATS DE COMANDA 1, DEMANDA DE CUADRATS PER COMANDA 1
OUT COMP_QUA1  ; COMPARA QUADRATS COM1
; rung 23
LDNOT HMI_C1_COM1_OK  ; VALIDACIO COM 1
@MOV(021) #0 C1_HMI_COM1_QUA  ; ENVIA EL ESTAT DE CUADRATS DE COMANDA 1
; rung 24: COMANDA 2 CUA
LD C1_E_F1  ; Produccio normal
OR C1_E_A2  ; Parada solicitud final de cicle
AND C1_EA_7  ; Etapa automatica DET4
AND EVA_CUADRAT  ; Foto per EVA=CUADRAT
ANDNOT COMP_QUA2  ; COMPARA QUADRATS COM2
AND COMP_QUA1  ; COMPARA QUADRATS COM1
LD C1_EA_42  ; FI CICLE
OR C1_E_D1  ; Parada de emergencia
OR P_First_Cycle
OR HMI_C1_Q_NO  ; RESPOSTA NEGATIVA A ACABAR CICLE
KEEP(011) C1_EA_20  ; COMANDA 2 CUADRAT ++
; rung 25
@LD C1_EA_20  ; COMANDA 2 CUADRAT ++
%LD C2_FI_CICLE
KEEP(011) CUA_COM2
; rung 26
LD CUA_COM2
@AND C2_FI_CICLE
++B(594) C1_HMI_COM2_QUA  ; ENVIA EL ESTAT DE CUADRAT DE COMANDA 2
; rung 27
LD P_On
AND=(300) C1_HMI_COM2_QUA HMI_COM2_CUA  ; ENVIA EL ESTAT DE CUADRAT DE COMANDA 2, DEMANDA DE CUADRATS PER COMANDA 2
OUT COMP_QUA2  ; COMPARA QUADRATS COM2

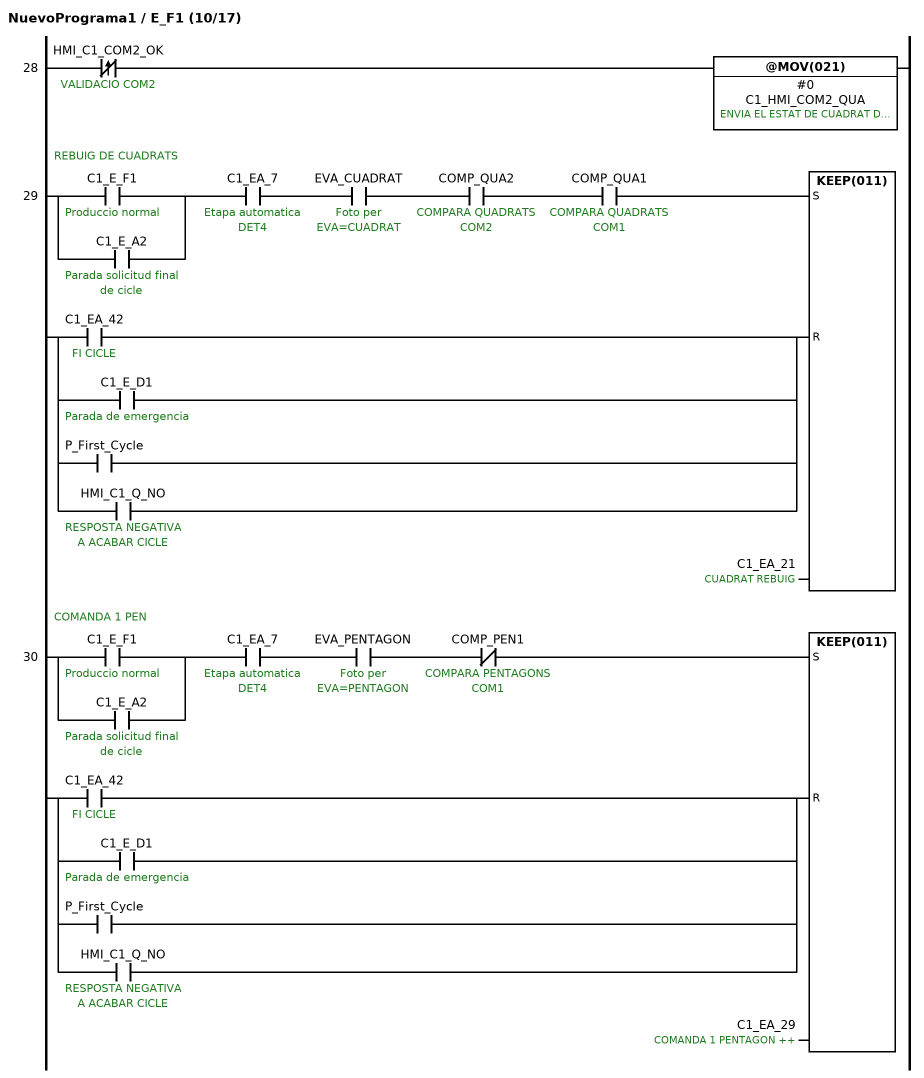
; rung 28
@LDNOT HMI_C1_COM2_OK  ; VALIDACIO COM2
@MOV(021) #0 C1_HMI_COM2_QUA  ; ENVIA EL ESTAT DE CUADRAT DE COMANDA 2
; rung 29: REBUIG DE CUADRATS
LD C1_E_F1  ; Produccio normal
OR C1_E_A2  ; Parada solicitud final de cicle
AND C1_EA_7  ; Etapa automatica DET4
AND EVA_CUADRAT  ; Foto per EVA=CUADRAT
AND COMP_QUA2  ; COMPARA QUADRATS COM2
AND COMP_QUA1  ; COMPARA QUADRATS COM1
LD C1_EA_42  ; FI CICLE
OR C1_E_D1  ; Parada de emergencia
OR P_First_Cycle
OR HMI_C1_Q_NO  ; RESPOSTA NEGATIVA A ACABAR CICLE
KEEP(011) C1_EA_21  ; CUADRAT REBUIG
; rung 30: COMANDA 1 PEN
LD C1_E_F1  ; Produccio normal
OR C1_E_A2  ; Parada solicitud final de cicle
AND C1_EA_7  ; Etapa automatica DET4
AND EVA_PENTAGON  ; Foto per EVA=PENTAGON
ANDNOT COMP_PEN1  ; COMPARA PENTAGONS COM1
LD C1_EA_42  ; FI CICLE
OR C1_E_D1  ; Parada de emergencia
OR P_First_Cycle
OR HMI_C1_Q_NO  ; RESPOSTA NEGATIVA A ACABAR CICLE
KEEP(011) C1_EA_29  ; COMANDA 1 PENTAGON ++

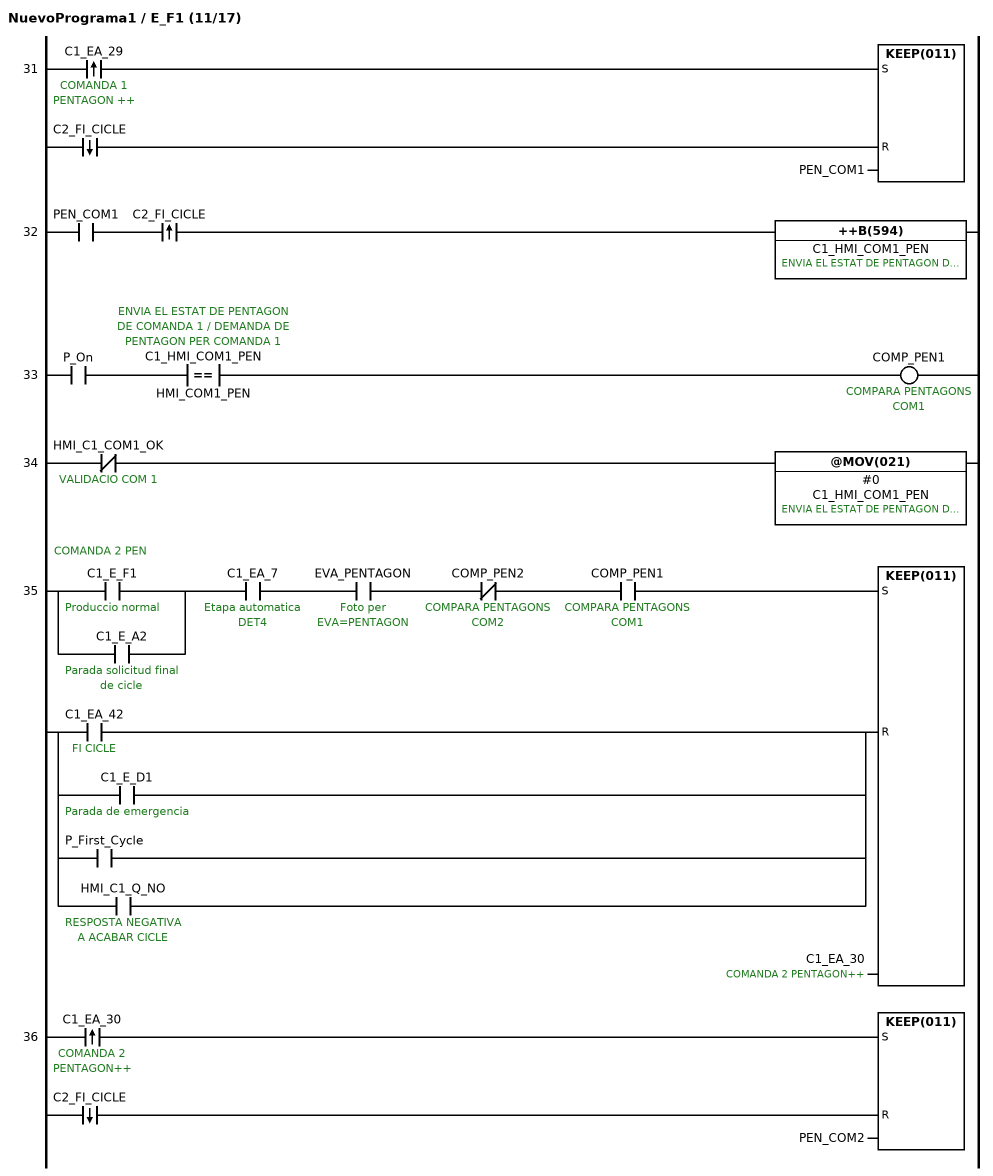
; rung 31
@LD C1_EA_29  ; COMANDA 1 PENTAGON ++
%LD C2_FI_CICLE
KEEP(011) PEN_COM1
; rung 32
LD PEN_COM1
@AND C2_FI_CICLE
++B(594) C1_HMI_COM1_PEN  ; ENVIA EL ESTAT DE PENTAGON DE COMANDA 1
; rung 33
LD P_On
AND=(300) C1_HMI_COM1_PEN HMI_COM1_PEN  ; ENVIA EL ESTAT DE PENTAGON DE COMANDA 1, DEMANDA DE PENTAGON PER COMANDA 1
OUT COMP_PEN1  ; COMPARA PENTAGONS COM1
; rung 34
LDNOT HMI_C1_COM1_OK  ; VALIDACIO COM 1
@MOV(021) #0 C1_HMI_COM1_PEN  ; ENVIA EL ESTAT DE PENTAGON DE COMANDA 1
; rung 35: COMANDA 2 PEN
LD C1_E_F1  ; Produccio normal
OR C1_E_A2  ; Parada solicitud final de cicle
AND C1_EA_7  ; Etapa automatica DET4
AND EVA_PENTAGON  ; Foto per EVA=PENTAGON
ANDNOT COMP_PEN2  ; COMPARA PENTAGONS COM2
AND COMP_PEN1  ; COMPARA PENTAGONS COM1
LD C1_EA_42  ; FI CICLE
OR C1_E_D1  ; Parada de emergencia
OR P_First_Cycle
OR HMI_C1_Q_NO  ; RESPOSTA NEGATIVA A ACABAR CICLE
KEEP(011) C1_EA_30  ; COMANDA 2 PENTAGON++
; rung 36
@LD C1_EA_30  ; COMANDA 2 PENTAGON++
%LD C2_FI_CICLE
KEEP(011) PEN_COM2

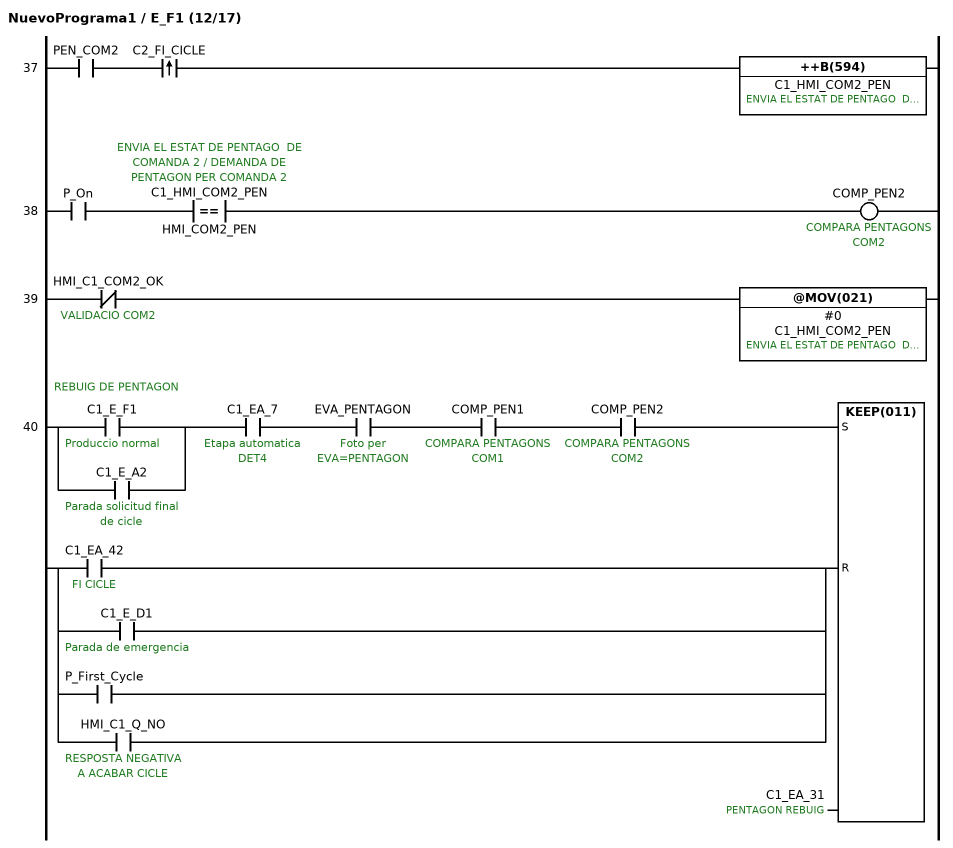
; rung 37
LD PEN_COM2
@AND C2_FI_CICLE
++B(594) C1_HMI_COM2_PEN  ; ENVIA EL ESTAT DE PENTAGO  DE COMANDA 2
; rung 38
LD P_On
AND=(300) C1_HMI_COM2_PEN HMI_COM2_PEN  ; ENVIA EL ESTAT DE PENTAGO  DE COMANDA 2, DEMANDA DE PENTAGON PER COMANDA 2
OUT COMP_PEN2  ; COMPARA PENTAGONS COM2
; rung 39
LDNOT HMI_C1_COM2_OK  ; VALIDACIO COM2
@MOV(021) #0 C1_HMI_COM2_PEN  ; ENVIA EL ESTAT DE PENTAGO  DE COMANDA 2
; rung 40: REBUIG DE PENTAGON
LD C1_E_F1  ; Produccio normal
OR C1_E_A2  ; Parada solicitud final de cicle
AND C1_EA_7  ; Etapa automatica DET4
AND EVA_PENTAGON  ; Foto per EVA=PENTAGON
AND COMP_PEN1  ; COMPARA PENTAGONS COM1
AND COMP_PEN2  ; COMPARA PENTAGONS COM2
LD C1_EA_42  ; FI CICLE
OR C1_E_D1  ; Parada de emergencia
OR P_First_Cycle
OR HMI_C1_Q_NO  ; RESPOSTA NEGATIVA A ACABAR CICLE
KEEP(011) C1_EA_31  ; PENTAGON REBUIG

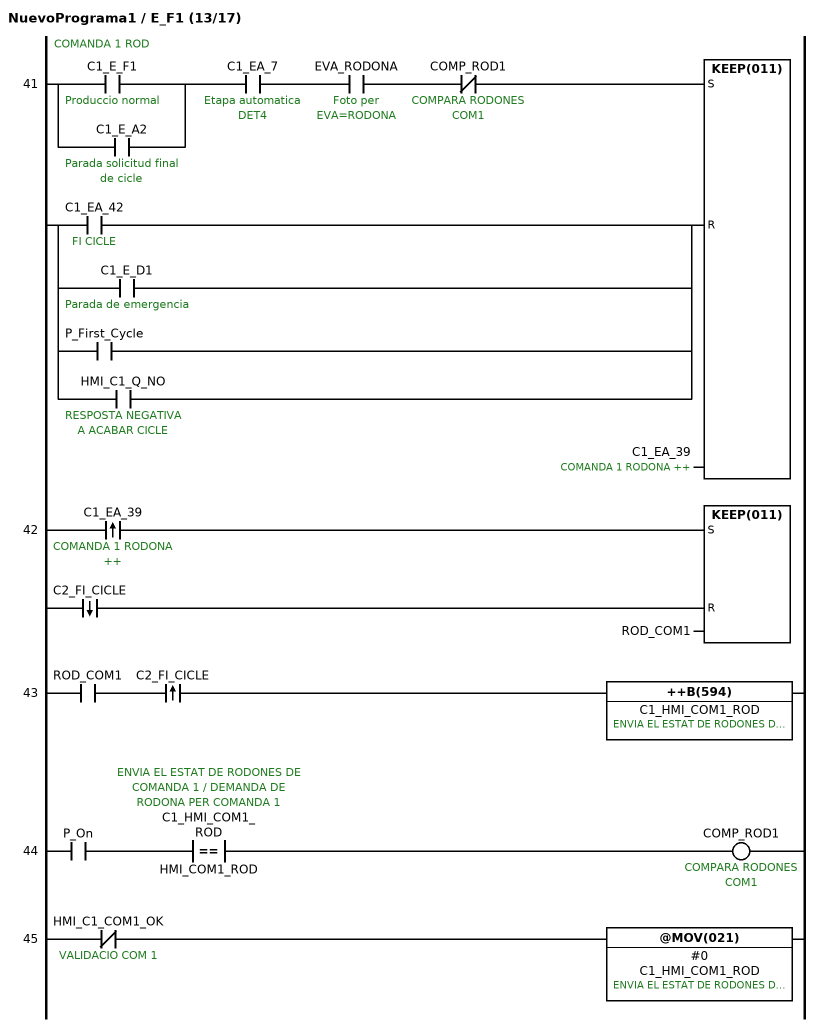
; rung 41: COMANDA 1 ROD
LD C1_E_F1  ; Produccio normal
OR C1_E_A2  ; Parada solicitud final de cicle
AND C1_EA_7  ; Etapa automatica DET4
AND EVA_RODONA  ; Foto per EVA=RODONA
ANDNOT COMP_ROD1  ; COMPARA RODONES COM1
LD C1_EA_42  ; FI CICLE
OR C1_E_D1  ; Parada de emergencia
OR P_First_Cycle
OR HMI_C1_Q_NO  ; RESPOSTA NEGATIVA A ACABAR CICLE
KEEP(011) C1_EA_39  ; COMANDA 1 RODONA ++
; rung 42
@LD C1_EA_39  ; COMANDA 1 RODONA ++
%LD C2_FI_CICLE
KEEP(011) ROD_COM1
; rung 43
LD ROD_COM1
@AND C2_FI_CICLE
++B(594) C1_HMI_COM1_ROD  ; ENVIA EL ESTAT DE RODONES DE COMANDA 1
; rung 44
LD P_On
AND=(300) C1_HMI_COM1_ROD HMI_COM1_ROD  ; ENVIA EL ESTAT DE RODONES DE COMANDA 1, DEMANDA DE RODONA PER COMANDA 1
OUT COMP_ROD1  ; COMPARA RODONES COM1
; rung 45
LDNOT HMI_C1_COM1_OK  ; VALIDACIO COM 1
@MOV(021) #0 C1_HMI_COM1_ROD  ; ENVIA EL ESTAT DE RODONES DE COMANDA 1

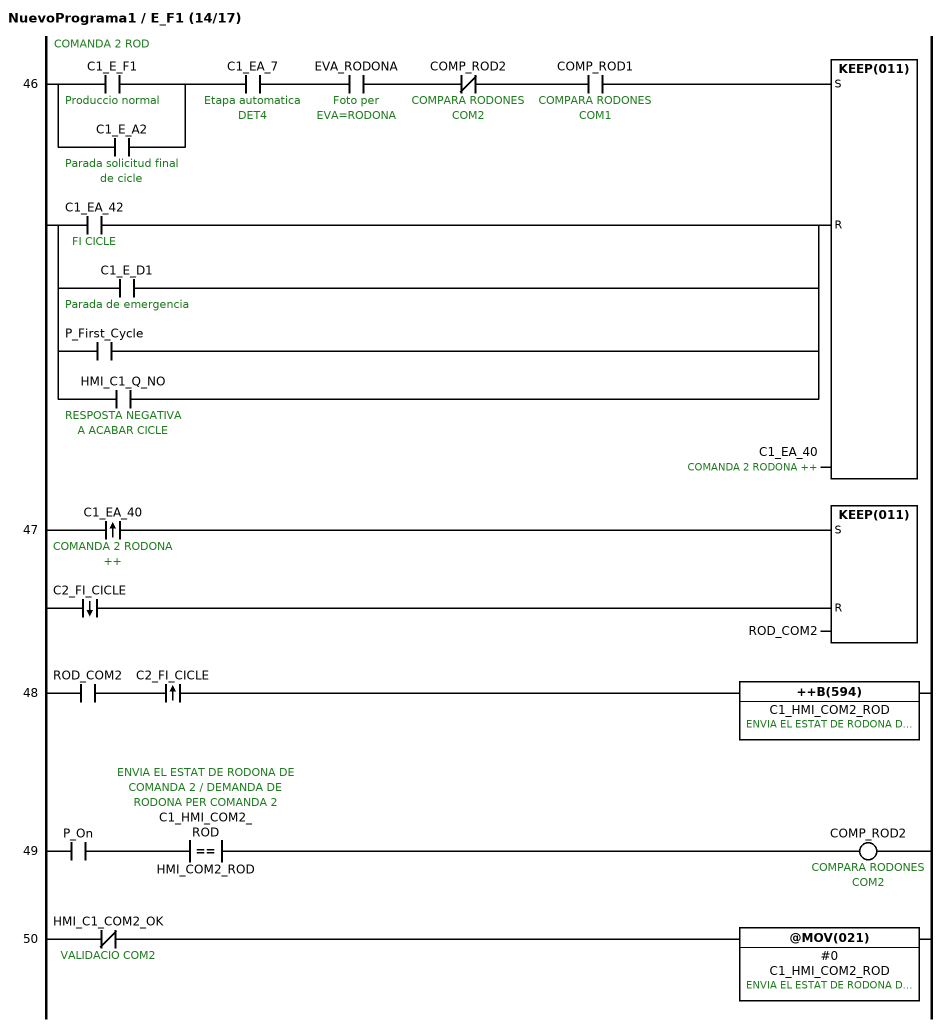
; rung 46: COMANDA 2 ROD
LD C1_E_F1  ; Produccio normal
OR C1_E_A2  ; Parada solicitud final de cicle
AND C1_EA_7  ; Etapa automatica DET4
AND EVA_RODONA  ; Foto per EVA=RODONA
ANDNOT COMP_ROD2  ; COMPARA RODONES COM2
AND COMP_ROD1  ; COMPARA RODONES COM1
LD C1_EA_42  ; FI CICLE
OR C1_E_D1  ; Parada de emergencia
OR P_First_Cycle
OR HMI_C1_Q_NO  ; RESPOSTA NEGATIVA A ACABAR CICLE
KEEP(011) C1_EA_40  ; COMANDA 2 RODONA ++
; rung 47
@LD C1_EA_40  ; COMANDA 2 RODONA ++
%LD C2_FI_CICLE
KEEP(011) ROD_COM2
; rung 48
LD ROD_COM2
@AND C2_FI_CICLE
++B(594) C1_HMI_COM2_ROD  ; ENVIA EL ESTAT DE RODONA DE COMANDA 2
; rung 49
LD P_On
AND=(300) C1_HMI_COM2_ROD HMI_COM2_ROD  ; ENVIA EL ESTAT DE RODONA DE COMANDA 2, DEMANDA DE RODONA PER COMANDA 2
OUT COMP_ROD2  ; COMPARA RODONES COM2
; rung 50
LDNOT HMI_C1_COM2_OK  ; VALIDACIO COM2
@MOV(021) #0 C1_HMI_COM2_ROD  ; ENVIA EL ESTAT DE RODONA DE COMANDA 2

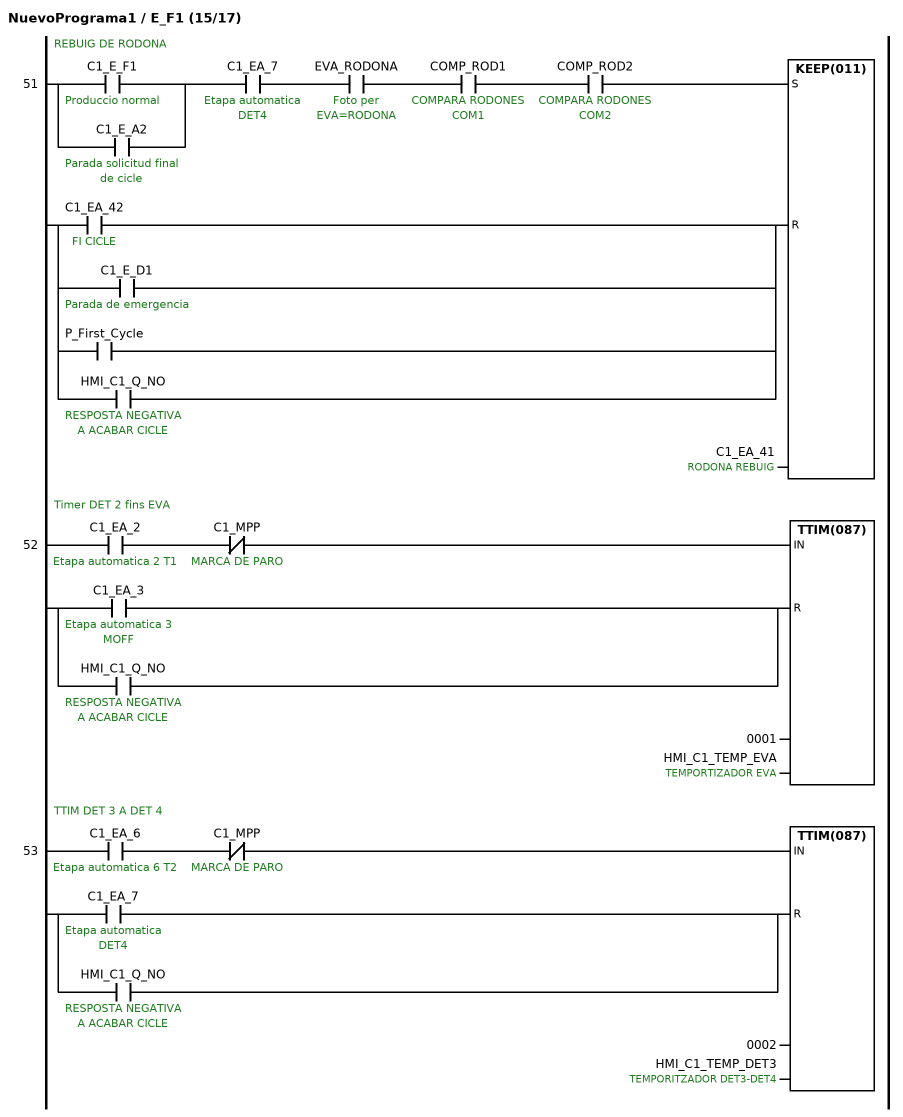
; rung 51: REBUIG DE RODONA
LD C1_E_F1  ; Produccio normal
OR C1_E_A2  ; Parada solicitud final de cicle
AND C1_EA_7  ; Etapa automatica DET4
AND EVA_RODONA  ; Foto per EVA=RODONA
AND COMP_ROD1  ; COMPARA RODONES COM1
AND COMP_ROD2  ; COMPARA RODONES COM2
LD C1_EA_42  ; FI CICLE
OR C1_E_D1  ; Parada de emergencia
OR P_First_Cycle
OR HMI_C1_Q_NO  ; RESPOSTA NEGATIVA A ACABAR CICLE
KEEP(011) C1_EA_41  ; RODONA REBUIG
; rung 52: Timer DET 2 fins EVA
LD C1_EA_2  ; Etapa automatica 2 T1
ANDNOT C1_MPP  ; MARCA DE PARO
LD C1_EA_3  ; Etapa automatica 3 MOFF
OR HMI_C1_Q_NO  ; RESPOSTA NEGATIVA A ACABAR CICLE
TTIM(087) 0001 HMI_C1_TEMP_EVA  ; TEMPORTIZADOR EVA
; rung 53: TTIM DET 3 A DET 4
LD C1_EA_6  ; Etapa automatica 6 T2
ANDNOT C1_MPP  ; MARCA DE PARO
LD C1_EA_7  ; Etapa automatica DET4
OR HMI_C1_Q_NO  ; RESPOSTA NEGATIVA A ACABAR CICLE
TTIM(087) 0002 HMI_C1_TEMP_DET3  ; TEMPORITZADOR DET3-DET4

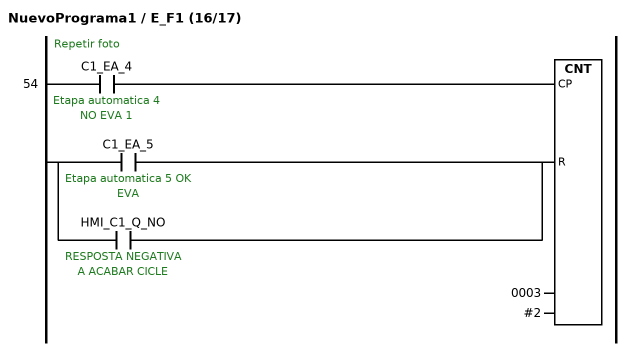
; rung 54: Repetir foto
LD C1_EA_4  ; Etapa automatica 4 NO EVA 1
LD C1_EA_5  ; Etapa automatica 5 OK EVA
OR HMI_C1_Q_NO  ; RESPOSTA NEGATIVA A ACABAR CICLE
CNT 0003 #2

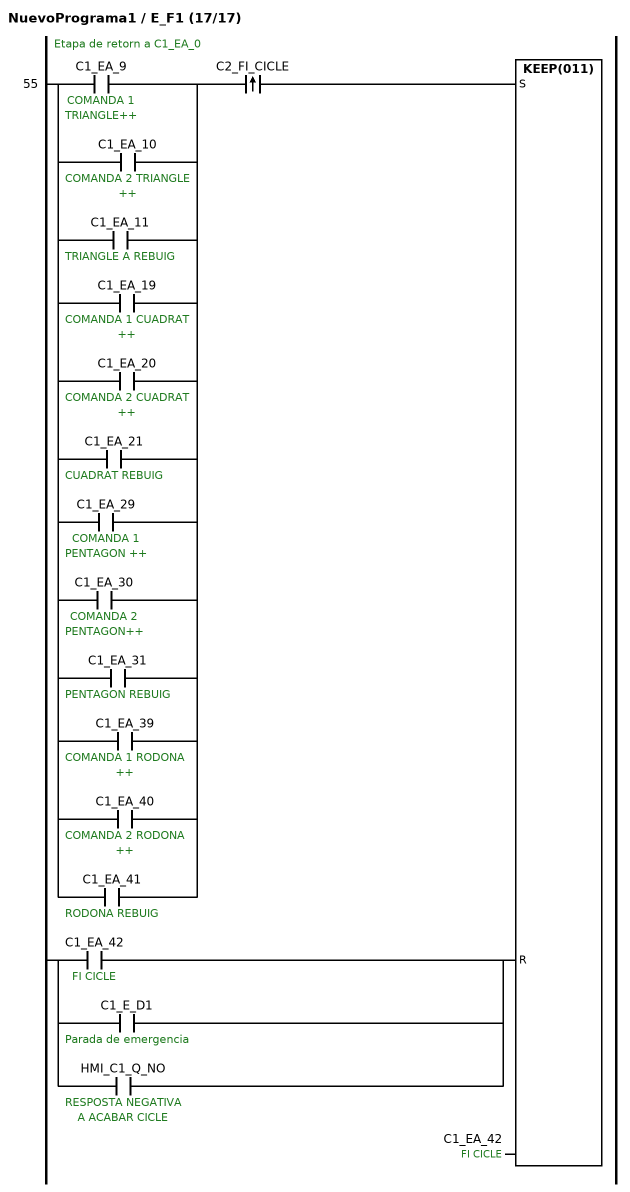
; rung 55: Etapa de retorn a C1_EA_0
LD C1_EA_9  ; COMANDA 1 TRIANGLE++
OR C1_EA_10  ; COMANDA 2 TRIANGLE ++
OR C1_EA_11  ; TRIANGLE A REBUIG
OR C1_EA_19  ; COMANDA 1 CUADRAT ++
OR C1_EA_20  ; COMANDA 2 CUADRAT ++
OR C1_EA_21  ; CUADRAT REBUIG
OR C1_EA_29  ; COMANDA 1 PENTAGON ++
OR C1_EA_30  ; COMANDA 2 PENTAGON++
OR C1_EA_31  ; PENTAGON REBUIG
OR C1_EA_39  ; COMANDA 1 RODONA ++
OR C1_EA_40  ; COMANDA 2 RODONA ++
OR C1_EA_41  ; RODONA REBUIG
@AND C2_FI_CICLE
LD C1_EA_42  ; FI CICLE
OR C1_E_D1  ; Parada de emergencia
OR HMI_C1_Q_NO  ; RESPOSTA NEGATIVA A ACABAR CICLE
KEEP(011) C1_EA_42  ; FI CICLE

### Section E_F4

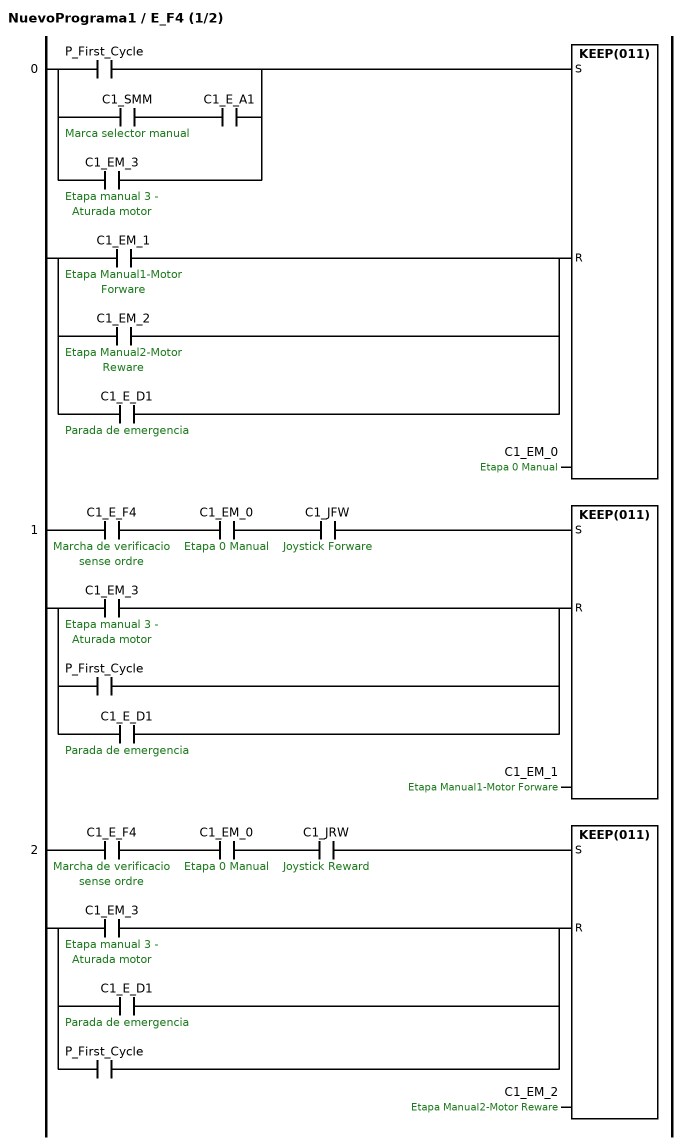
; rung 0
LD P_First_Cycle
LD C1_SMM  ; Marca selector manual
AND C1_E_A1
ORLD
OR C1_EM_3  ; Etapa manual 3 - Aturada motor
LD C1_EM_1  ; Etapa Manual1-Motor Forware
OR C1_EM_2  ; Etapa Manual2-Motor Reware
OR C1_E_D1  ; Parada de emergencia
KEEP(011) C1_EM_0  ; Etapa 0 Manual
; rung 1
LD C1_E_F4  ; Marcha de verificacio sense ordre
AND C1_EM_0  ; Etapa 0 Manual
AND C1_JFW  ; Joystick Forware
LD C1_EM_3  ; Etapa manual 3 - Aturada motor
OR P_First_Cycle
OR C1_E_D1  ; Parada de emergencia
KEEP(011) C1_EM_1  ; Etapa Manual1-Motor Forware
; rung 2
LD C1_E_F4  ; Marcha de verificacio sense ordre
AND C1_EM_0  ; Etapa 0 Manual
AND C1_JRW  ; Joystick Reward
LD C1_EM_3  ; Etapa manual 3 - Aturada motor
OR C1_E_D1  ; Parada de emergencia
OR P_First_Cycle
KEEP(011) C1_EM_2  ; Etapa Manual2-Motor Reware

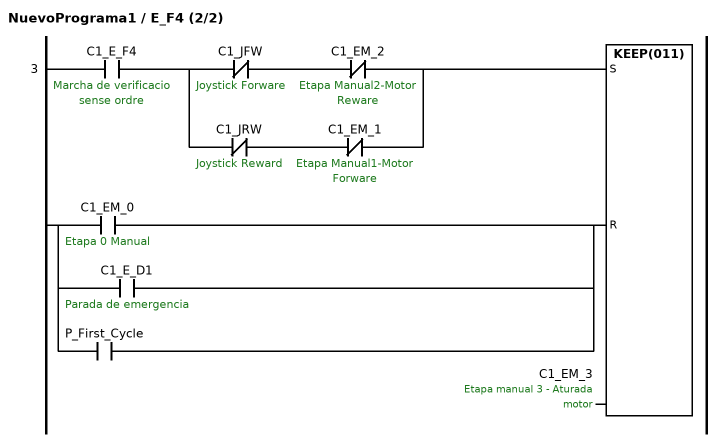
; rung 3
LD C1_E_F4  ; Marcha de verificacio sense ordre
LDNOT C1_JFW  ; Joystick Forware
ANDNOT C1_EM_2  ; Etapa Manual2-Motor Reware
LDNOT C1_JRW  ; Joystick Reward
ANDNOT C1_EM_1  ; Etapa Manual1-Motor Forware
ORLD
ANDLD
LD C1_EM_0  ; Etapa 0 Manual
OR C1_E_D1  ; Parada de emergencia
OR P_First_Cycle
KEEP(011) C1_EM_3  ; Etapa manual 3 - Aturada motor

### Section ACCIONS

